VAR_GLOBAL CONSTANT
	TAMANO_LISTA_PIEZAS : UINT := 8;
	TAMANO_LISTA_CONDICIONES : UINT := 6;
END_VAR

(* stored: Version 1.1.0.1, ProductVersion 3.1.4024.15
   GVL Constantes: Id {86eafa11-8f6d-4d87-b4ab-83c07790114d} *)
